PROGRAM FunctionBlockMisc
VAR

	FB_WritePersistentData_0: FB_WritePersistentData;
	TON_0: TON;
	TON_1: TON;
	NotBusy: BOOL;
	//1 second ups function writes data and performs quick shutdown
	//check on input SPDM_VAR_BOOST - saves different task data on different PLC cycles?
	FB_S_UPS_BAPI_0: FB_S_UPS_BAPI; 
END_VAR

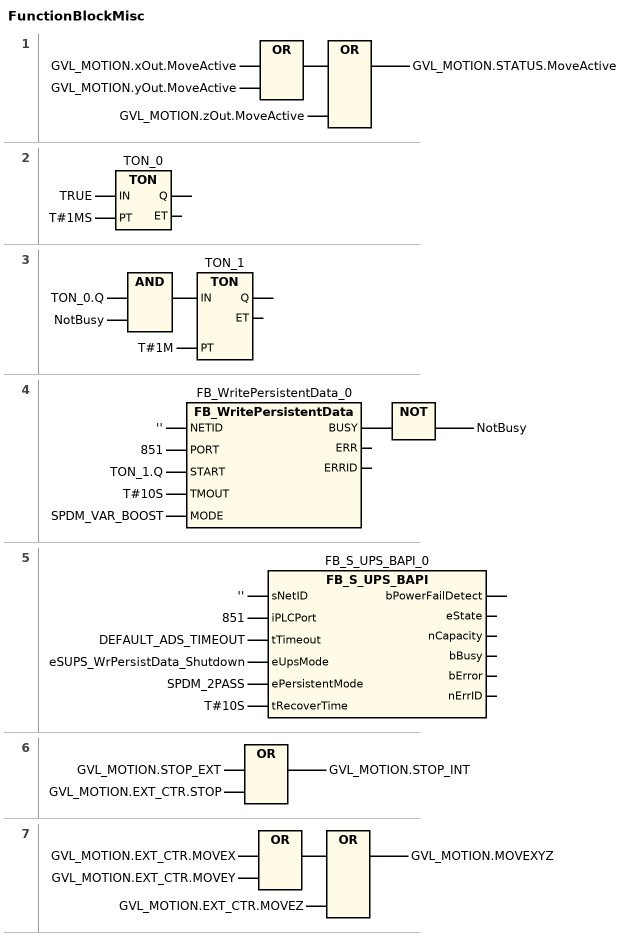
// NETWORK 1
GVL_MOTION.STATUS.MoveActive := (GVL_MOTION.xOut.MoveActive OR GVL_MOTION.yOut.MoveActive) OR GVL_MOTION.zOut.MoveActive;

// NETWORK 2
TON_0(IN := TRUE, PT := T#1MS); // TON

// NETWORK 3
TON_1(IN := TON_0.Q AND NotBusy, PT := T#1M); // TON

// NETWORK 4
FB_WritePersistentData_0(NETID := '', PORT := 851, START := TON_1.Q, TMOUT := T#10S, MODE := SPDM_VAR_BOOST); // FB_WritePersistentData
NotBusy := NOT FB_WritePersistentData_0.BUSY;

// NETWORK 5
FB_S_UPS_BAPI_0(
    sNetID := '',
    iPLCPort := 851,
    tTimeout := DEFAULT_ADS_TIMEOUT,
    eUpsMode := eSUPS_WrPersistData_Shutdown,
    ePersistentMode := SPDM_2PASS,
    tRecoverTime := T#10S); // FB_S_UPS_BAPI

// NETWORK 6
GVL_MOTION.STOP_INT := GVL_MOTION.STOP_EXT OR GVL_MOTION.EXT_CTR.STOP;

// NETWORK 7
GVL_MOTION.MOVEXYZ := (GVL_MOTION.EXT_CTR.MOVEX OR GVL_MOTION.EXT_CTR.MOVEY) OR GVL_MOTION.EXT_CTR.MOVEZ;

END_PROGRAM

(* stored: Version 1.1.0.1, ProductVersion 3.1.4026.18
   POU FunctionBlockMisc: Id {3268ba04-f1cd-44f6-8ab5-5ffeb5291a7a}, SpecialFunc None *)
